TYPE DUT_CS_Motor_Freq EXTENDS DUT_Com_Base_Motor_Freq :
STRUCT
	Interlock: BOOL; // Interlock CM
END_STRUCT
END_TYPE

(* stored: Version 1.1.0.1, ProductVersion 3.1.4024.12
   DUT DUT_CS_Motor_Freq: Id {4dad7a8e-baa2-475b-a7cd-25883465ef46} *)
